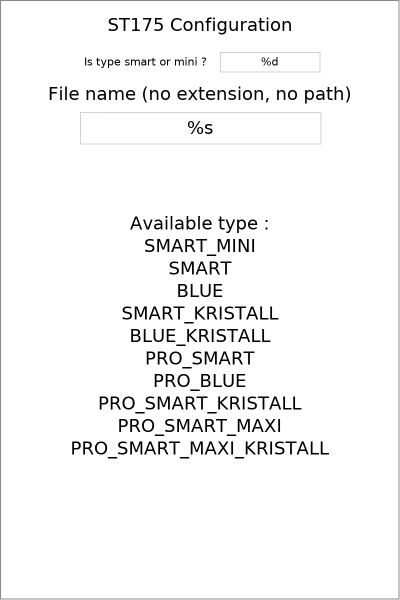
VISUALIZATION VISU_Recipe_ST175  // 400x600
    Textfield (80,112 241x32), "%s", text variable: _20_AUTO.recipe.st175.file_name
        OnMouseDown: write the text variable via Default
    Label (0,5 400x40), "ST175 Configuration"
    Label (24,84 352x20), "File name (no extension, no path)"
    Label (59,174 282x324), "Available type : SMART_MINI SMART BLUE SMART_KRISTALL BLUE_KRISTALL PRO_SMART PRO_BLUE PRO_SMART_KRISTALL PRO_SMART_MAXI PRO_SMART_MAXI_KRISTALL"
    Textfield (220,52 100x20), "%d", text variable: _20_AUTO.recipe.st175.isTypeSmartOrMini
        OnMouseDown: write the text variable via Default
    Label (10,52 200x20), "Is type smart or mini ?"
END_VISUALIZATION

(* stored: Version 1.1.0.1, ProductVersion 3.1.4024.6
   Visu VISU_Recipe_ST175: Id {9bcd3d30-c5e5-480c-a76b-bccd1c299c77} *)
